(* CODESYS project Pizzaprocessor_03_11_2025.export

Project tree, tasks and I/O mapping:
  Device : CODESYS Control Win V3 x64, CODESYS, version 3.5.21.10
    application Application
      libraries: Standard, 3.5.18.0 (System)
      task MainTask (cyclic, interval t#20ms, priority 1) calls Supervisor_PRG
      Communication Manager
        OPC UA Server
          IEC Symbol Publishing
          Symbol Set
      data type ConveyorStatus
      data type HopperStatus
      global variables Global_Variables
      function block FB_Conveyor [ST]
      function block FB_Hopper [ST]
      program Supervisor_PRG [ST]
*)

// Device/Application/ConveyorStatus
TYPE ConveyorStatus :
STRUCT
	Conveyor_ID: INT; // Conveyor number/ID
	Speed: REAL; // Percentage of speed
	Jam_Detected: BOOL; //Conveyor is Jammed
	Running: BOOL;
	
END_STRUCT
END_TYPE

// Device/Application/HopperStatus
TYPE HopperStatus :
STRUCT
	Hopper_Id: INT; //id for each Hopper
	Fill_Level: REAL; //percentage of hooper
	Ingredient_ID: STRING(20); //Ingredient Name
	Alarm_Active: BOOL; //Alarm
	Is_Dispensing: BOOL;//Ingredient is being dispensed
END_STRUCT
END_TYPE

// Device/Application/Global_Variables
{attribute 'qualified_only'}
VAR_GLOBAL
END_VAR

// Device/Application/Supervisor_PRG
PROGRAM Supervisor_PRG
VAR
	//Mode Control
	b_Mode: BOOL; //True = Auto, False = Manual

	//Status from Sensor
	b_Hopper_Empty:ARRAY[1..5] OF BOOL; // 1=Base, 2=Toppings, 3=Oregano, 4=Chilli, 5=Box (if you treat Box similarly)
	b_Conveyor_Jam: ARRAY [1..3] OF BOOL; //3 conveyors Jam Status

	//Process Flags
	 // Interlocks for hoppers or zones (e.g., 1=Base Hopper, 2=Toppings Hopper, etc.)
    b_Interlock_Hopper: ARRAY[1..5] OF BOOL;  // Matches hopper indices
    // Interlocks for conveyors
    b_Interlock_Conveyor: ARRAY[1..3] OF BOOL;
    // Interlocks for other zones like Heating, Packing - separate BOOLs or an array
    b_Interlock_OtherZones: ARRAY[1..2] OF BOOL; // Example: 1=HeatingZone, 2=PackingStation


	 // Alarm Flags
    b_Alarm_HopperEmpty : BOOL;
    b_Alarm_ConveyorJam : BOOL;
	
	

    // Identifier
    i_Jammed_Conveyor_Index : INT;    // 0 = none, else 1..n conveyor index
    i_Empty_Hopper_Index: INT;
    // Alarm Reset Command
    b_Alarm_Reset_Command : BOOL;      // Command from HMI to reset alarms
	
		
END_VAR

END_PROGRAM

// Device/Application/FB_Conveyor
FUNCTION_BLOCK FB_Conveyor
VAR_INPUT
	Start: BOOL;
	Speed_Setpoint: REAL; //percentage in speed
END_VAR
VAR_OUTPUT
	Running: BOOL; //
	Fault: BOOL; //
	Jam_Detected: BOOL; //
	Current_Speed: REAL; //
END_VAR

VAR
	State: INT; //0=Ideal, 1=running, 2=Fault
END_VAR

// Logic Framework
IF Fault THEN
	Running := FALSE;
	Current_Speed := 0.0;
	State := 2;
ELSE
	IF NOT Fault AND Start = TRUE THEN
	   Running := TRUE;
	   Current_Speed := Speed_Setpoint;
	   State := 1;
	 ELSIF NOT Start THEN 
     	Running := FALSE;
	    Current_Speed := 0.0;
	    State := 0;	
		 
		
		
	END_IF
	
END_IF

END_FUNCTION_BLOCK

// Device/Application/FB_Hopper
FUNCTION_BLOCK FB_Hopper
VAR_INPUT
	StartDispense: BOOL;
	StopDispense:BOOL;
END_VAR
VAR_OUTPUT
	Status:HopperStatus;
END_VAR
VAR Internal_State: BOOL; // False=Idle True= Dispensing
END_VAR

//Hopper Control Logic
IF StartDispense THEN
	Status.Is_Dispensing:= TRUE;
	Internal_State := TRUE;
ELSIF StopDispense THEN
	Status.Is_Dispensing:= FALSE;
	Internal_State := FALSE;
END_IF

//Simulate Ingredient level
IF Internal_State =1 THEN
   Status.Fill_Level := Status.Fill_Level - 0.1; // Decrement per Order
END_IF

//Alarm Logic
status.Alarm_Active := (status.Fill_Level < 5.0);

END_FUNCTION_BLOCK
